FUNCTION_BLOCK CachedComp IMPLEMENTS I_Debug
VAR_INPUT
END_VAR
VAR_OUTPUT
END_VAR
VAR
END_VAR

//FB_Init is always available implicitly and it is used primarily for initialization.
//The return value is not evaluated. For a specific influence, you can also declare the
//methods explicitly and provide additional code there with the standard initialization
//code. You can evaluate the return value.
METHOD FB_Init: BOOL
VAR_INPUT
    bInitRetains: BOOL; // TRUE: the retain variables are initialized (reset warm / reset cold)
    bInCopyCode: BOOL;  // TRUE: the instance will be copied to the copy code afterward (online change)

	iComponent	: I_Component;
	iRegister	: I_MutCompRegister;
	refCache	: REFERENCE TO UDINT;
END_VAR
VAR
	_eResult	: Result;
END_VAR
IF iRegister = 0 THEN
	DebugMsg(THIS^, 'iRegister = 0!');
	RETURN;
END_IF

IF __ISVALIDREF(refCache) THEN
	IF refCache = 0 THEN
		refCache := refCache;
	ELSE
		DebugMsg(THIS^, 'refCache is already assigned!');
	END_IF
ELSE
	DebugMsg(THIS^, 'refCache is invalid!');
END_IF

IF IsErr(iRegister.Insert(iComponent), eCarry => _eResult) THEN
	DebugMsg(THIS^, Tc2_Standard.CONCAT('I_MutCompRegister.Insert(iComponent) failed with code: ', TO_STRING(_eResult)));
END_IF
END_METHOD

END_FUNCTION_BLOCK

(* stored: Version 1.1.0.1
   POU CachedComp: Id {24ffeaed-00ab-44d1-9e0c-e416509d8090}, SpecialFunc None
   Method Fb_init: Id {a3ffd9c0-b369-4f73-b509-0eeb5b55cffd} *)
